FUNCTION_BLOCK Recipe_10058_RedOne
VAR_INPUT
	execute: BOOL;
	Order: DUT_RECIPEORDER;
END_VAR
VAR_OUTPUT
	RecipeInfo: DUT_RECIPEOFFER;
	RecipeDone: BOOL;
	InitDone: BOOL;
	Ready: BOOL;
END_VAR
VAR
	userparametersum: LREAL;
	StepDone: BOOL;
	i: INT;
	Command: ARRAY[1..5] OF DUT_RecipeCommand;
	NextSkill: BOOL;
	SectionReady: BOOL;
END_VAR

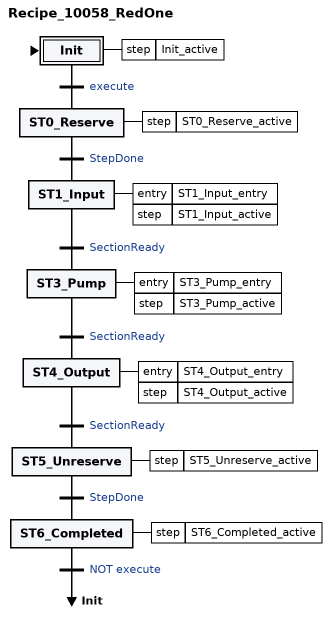
INITIAL_STEP Init:
    Init_active(N);  // step action
END_STEP
TRANSITION FROM Init TO ST0_Reserve
    := execute;
END_TRANSITION
STEP ST0_Reserve:
    ST0_Reserve_active(N);  // step action
END_STEP
TRANSITION FROM ST0_Reserve TO ST1_Input
    := StepDone;
END_TRANSITION
STEP ST1_Input:
    ST1_Input_entry(P1);  // entry action
    ST1_Input_active(N);  // step action
END_STEP
TRANSITION FROM ST1_Input TO ST3_Pump
    := SectionReady;
END_TRANSITION
STEP ST3_Pump:
    ST3_Pump_entry(P1);  // entry action
    ST3_Pump_active(N);  // step action
END_STEP
TRANSITION FROM ST3_Pump TO ST4_Output
    := SectionReady;
END_TRANSITION
STEP ST4_Output:
    ST4_Output_entry(P1);  // entry action
    ST4_Output_active(N);  // step action
END_STEP
TRANSITION FROM ST4_Output TO ST5_Unreserve
    := SectionReady;
END_TRANSITION
STEP ST5_Unreserve:
    ST5_Unreserve_active(N);  // step action
END_STEP
TRANSITION FROM ST5_Unreserve TO ST6_Completed
    := StepDone;
END_TRANSITION
STEP ST6_Completed:
    ST6_Completed_active(N);  // step action
END_STEP
TRANSITION FROM ST6_Completed TO Init
    := NOT execute;
END_TRANSITION

ACTION ST14_Exit_active:
SectionReady := TRUE;
END_ACTION

ACTION ST12_Input_active:
//RT: 2014.11.23: Input Modul auslösen
StepDone := FALSE;

//Skill auswählen
ExecuteSkill.SkillID 		:= 1402;
ExecuteSkill.SkillName	 	:= 'Input';

//Parameter setzen

ExecuteSkill.Parameter[1].ID := 1;
ExecuteSkill.Parameter[1].Name := 'TaskID';
ExecuteSkill.Parameter[1].Value := Order.TaskID;


(*
ExecuteSkill.Parameter[2].ID := ;
ExecuteSkill.Parameter[2].Name := '';
ExecuteSkill.Parameter[2].Value := ;
*)

(*
ExecuteSkill.Parameter[3].ID := ;
ExecuteSkill.Parameter[3].Name := '';
ExecuteSkill.Parameter[3].Value := ;
*)

(*
ExecuteSkill.Parameter[4].ID := ;
ExecuteSkill.Parameter[4].Name := '';
ExecuteSkill.Parameter[4].Value := ;
*)

(*
ExecuteSkill.Parameter[5].ID := ;
ExecuteSkill.Parameter[5].Name := '';
ExecuteSkill.Parameter[5].Value := ;
*)



ExecuteSkill();

StepDone := ExecuteSkill.Done;
END_ACTION

ACTION ST34_Exit_active:
SectionReady := TRUE;
END_ACTION

ACTION ST41_BlockOutput_active:
//RT: 2014.11.23: Blockirt den Mover an Position
StepDone := FALSE;

//Skill auswählen
ExecuteSkill.SkillID 		:= 1315;
ExecuteSkill.SkillName	 	:= 'Block';

//Parameter setzen

ExecuteSkill.Parameter[1].ID := 1;
ExecuteSkill.Parameter[1].Name := 'TaskID';
ExecuteSkill.Parameter[1].Value := Order.TaskID;


(*
ExecuteSkill.Parameter[2].ID := ;
ExecuteSkill.Parameter[2].Name := '';
ExecuteSkill.Parameter[2].Value := ;
*)

(*
ExecuteSkill.Parameter[3].ID := ;
ExecuteSkill.Parameter[3].Name := '';
ExecuteSkill.Parameter[3].Value := ;
*)

(*
ExecuteSkill.Parameter[4].ID := ;
ExecuteSkill.Parameter[4].Name := '';
ExecuteSkill.Parameter[4].Value := ;
*)

(*
ExecuteSkill.Parameter[5].ID := ;
ExecuteSkill.Parameter[5].Name := '';
ExecuteSkill.Parameter[5].Value := ;
*)



ExecuteSkill();

StepDone := ExecuteSkill.Done;
END_ACTION

ACTION ST13_UnblockInput_active:
//RT: 2014.11.23: Gibt Mover Position Frei
StepDone := FALSE;

//Skill auswählen
ExecuteSkill.SkillID 		:= 1316;
ExecuteSkill.SkillName	 	:= 'Unblock';

//Parameter setzen

ExecuteSkill.Parameter[1].ID := 1;
ExecuteSkill.Parameter[1].Name := 'TaskID';
ExecuteSkill.Parameter[1].Value := Order.TaskID;


(*
ExecuteSkill.Parameter[2].ID := ;
ExecuteSkill.Parameter[2].Name := '';
ExecuteSkill.Parameter[2].Value := ;
*)

(*
ExecuteSkill.Parameter[3].ID := ;
ExecuteSkill.Parameter[3].Name := '';
ExecuteSkill.Parameter[3].Value := ;
*)

(*
ExecuteSkill.Parameter[4].ID := ;
ExecuteSkill.Parameter[4].Name := '';
ExecuteSkill.Parameter[4].Value := ;
*)

(*
ExecuteSkill.Parameter[5].ID := ;
ExecuteSkill.Parameter[5].Name := '';
ExecuteSkill.Parameter[5].Value := ;
*)



ExecuteSkill();

StepDone := ExecuteSkill.Done;
END_ACTION

ACTION ST4_Output_active:
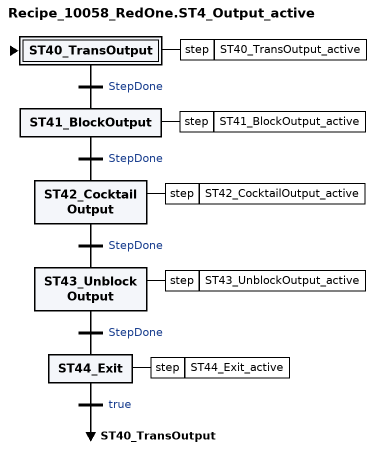
INITIAL_STEP ST40_TransOutput:
    ST40_TransOutput_active(N);  // step action
END_STEP
TRANSITION FROM ST40_TransOutput TO ST41_BlockOutput
    := StepDone;
END_TRANSITION
STEP ST41_BlockOutput:
    ST41_BlockOutput_active(N);  // step action
END_STEP
TRANSITION FROM ST41_BlockOutput TO ST42_CocktailOutput
    := StepDone;
END_TRANSITION
STEP ST42_CocktailOutput:
    ST42_CocktailOutput_active(N);  // step action
END_STEP
TRANSITION FROM ST42_CocktailOutput TO ST43_UnblockOutput
    := StepDone;
END_TRANSITION
STEP ST43_UnblockOutput:
    ST43_UnblockOutput_active(N);  // step action
END_STEP
TRANSITION FROM ST43_UnblockOutput TO ST44_Exit
    := StepDone;
END_TRANSITION
STEP ST44_Exit:
    ST44_Exit_active(N);  // step action
END_STEP
TRANSITION FROM ST44_Exit TO ST40_TransOutput
    := true;
END_TRANSITION
END_ACTION

ACTION ST42_CocktailOutput_active:
//RT: 2014.11.23: Ausgeben des Produktes
StepDone := FALSE;

//Skill auswählen
ExecuteSkill.SkillID 		:= 1403;
ExecuteSkill.SkillName	 	:= 'Output';

//Parameter setzen

ExecuteSkill.Parameter[1].ID := 1;
ExecuteSkill.Parameter[1].Name := 'TaskID';
ExecuteSkill.Parameter[1].Value := Order.TaskID;


(*
ExecuteSkill.Parameter[2].ID := ;
ExecuteSkill.Parameter[2].Name := '';
ExecuteSkill.Parameter[2].Value := ;
*)

(*
ExecuteSkill.Parameter[3].ID := ;
ExecuteSkill.Parameter[3].Name := '';
ExecuteSkill.Parameter[3].Value := ;
*)

(*
ExecuteSkill.Parameter[4].ID := ;
ExecuteSkill.Parameter[4].Name := '';
ExecuteSkill.Parameter[4].Value := ;
*)

(*
ExecuteSkill.Parameter[5].ID := ;
ExecuteSkill.Parameter[5].Name := '';
ExecuteSkill.Parameter[5].Value := ;
*)



ExecuteSkill();

StepDone := ExecuteSkill.Done;
END_ACTION

ACTION ST40_TransOutput_active:
//RT: 2014.11.23: Mover zum Output
StepDone := FALSE;

//Skill auswählen
ExecuteSkill.SkillID 		:= 1320;
ExecuteSkill.SkillName	 	:= 'Transport';

//Parameter setzen

ExecuteSkill.Parameter[3].ID := 3;
ExecuteSkill.Parameter[3].Name := 'Velocity';
ExecuteSkill.Parameter[3].Value := 300;



ExecuteSkill.Parameter[1].ID :=  1;
ExecuteSkill.Parameter[1].Name := 'TargetPosition X';
ExecuteSkill.Parameter[1].Value := 30 ;
ExecuteSkill.Parameter[1].StringValue := '#DP#2#XPosition';



ExecuteSkill.Parameter[2].ID := 2;
ExecuteSkill.Parameter[2].Name := 'TargetPosition Z';
ExecuteSkill.Parameter[2].Value := 100;// ZCookieModule - ZCookieModuleCalibration - 2* Cookiethickness + toppingthickness+ Preasureheight  ;



(* ExecuteSkill.Parameter[4].ID := 4;
ExecuteSkill.Parameter[4].Name := 'Acceleration';
ExecuteSkill.Parameter[4].Value :=0 ;

*)
(*
ExecuteSkill.Parameter[5].ID := ;
ExecuteSkill.Parameter[5].Name := '';
ExecuteSkill.Parameter[5].Value := ;
*)



ExecuteSkill();

StepDone := ExecuteSkill.Done;
END_ACTION

ACTION ST3_Pump_active:
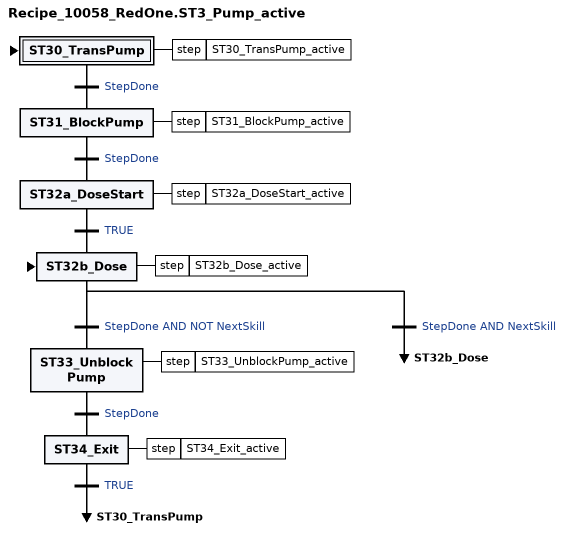
INITIAL_STEP ST30_TransPump:
    ST30_TransPump_active(N);  // step action
END_STEP
TRANSITION FROM ST30_TransPump TO ST31_BlockPump
    := StepDone;
END_TRANSITION
STEP ST31_BlockPump:
    ST31_BlockPump_active(N);  // step action
END_STEP
TRANSITION FROM ST31_BlockPump TO ST32a_DoseStart
    := StepDone;
END_TRANSITION
STEP ST32a_DoseStart:
    ST32a_DoseStart_active(N);  // step action
END_STEP
TRANSITION FROM ST32a_DoseStart TO ST32b_Dose
    := TRUE;
END_TRANSITION
STEP ST32b_Dose:
    ST32b_Dose_active(N);  // step action
END_STEP
TRANSITION FROM ST32b_Dose TO ST33_UnblockPump
    := StepDone AND NOT NextSkill;
END_TRANSITION
STEP ST33_UnblockPump:
    ST33_UnblockPump_active(N);  // step action
END_STEP
TRANSITION FROM ST33_UnblockPump TO ST34_Exit
    := StepDone;
END_TRANSITION
STEP ST34_Exit:
    ST34_Exit_active(N);  // step action
END_STEP
TRANSITION FROM ST34_Exit TO ST30_TransPump
    := TRUE;
END_TRANSITION
TRANSITION FROM ST32b_Dose TO ST32b_Dose
    := StepDone AND NextSkill;
END_TRANSITION
END_ACTION

ACTION ST32a_DoseStart_active:
//RT: 2014.11.23: Summe aller zutaten zum Normiren

userparametersum := 0;
FOR i := 1 TO UserParameterCnt DO
	IF NOT (order.UserParameter[i].Value = 0) THEN
		userparametersum := userparametersum + order.UserParameter[i].Value;
	
	END_IF
END_FOR
IF userparametersum = 0 THEN
userparametersum := -1;
END_IF

//RT: 2014.11.23: Start wert des Arrays setzen
i := 1;
NextSkill := TRUE ;
END_ACTION

ACTION Init_active:
//RT: 2014.11.23: Vorbereiten der daten und der HMI
RecipeDone := FALSE;

// Initialisation of Recipe Parameters an name etc
RecipeInfo.Name := 'Red One';
RecipeInfo.Description := '';
RecipeInfo.Dummy := FALSE;
RecipeInfo.RecipeID := 10058; 	// 
Initdone := TRUE;

//RT: 2014.11.23: wenn weniger als 5 alle lehren skills SkillID := 0
Command[1].SkillID := 1117;
Command[1].SkillName := 'Orange Juice';
Command[1].Quantity := 41;

Command[2].SkillID := 1112;
Command[2].SkillName := 'Lemon Juice';
Command[2].Quantity := 8;

Command[3].SkillID := 1114;
Command[3].SkillName := 'Pineapple Juice';
Command[3].Quantity := 41;

Command[4].SkillID := 1111;
Command[4].SkillName := 'Grenadine Syrup';
Command[4].Quantity := 8;

Command[5].SkillID := 0;
Command[5].SkillName := 'Nothing';
Command[5].Quantity := 0;








//Parameter 0:

	RecipeInfo.UserParameter[0].Dummy 		:= FALSE;
	RecipeInfo.UserParameter[0].Default		:= 200;
	RecipeInfo.UserParameter[0].Description	:= 'Gives the total fluid amount in the glass';
	RecipeInfo.UserParameter[0].MaxValue	:= 200;
	RecipeInfo.UserParameter[0].MinValue	:= 10;
	RecipeInfo.UserParameter[0].Name		:= 'Total Liquid Amount';
	RecipeInfo.UserParameter[0].Unit		:= 'ml';
	
//Parameter 1-5:
FOR i := 1 TO 5 DO
	IF Command[i].SkillID = 0 THEN
		RecipeInfo.UserParameter[i].Dummy 		:= TRUE;
	ELSE
		RecipeInfo.UserParameter[i].Dummy 		:= FALSE;
		RecipeInfo.UserParameter[i].Default		:= Command[i].Quantity;
		RecipeInfo.UserParameter[i].Description	:= Command[i].SkillName;
		RecipeInfo.UserParameter[i].MaxValue	:= 100;
		RecipeInfo.UserParameter[i].MinValue	:= 1;
		RecipeInfo.UserParameter[i].Name		:= Command[i].SkillName;
		RecipeInfo.UserParameter[i].Unit		:= 'ml';	
	END_IF
END_FOR
END_ACTION

ACTION ST30_TransPump_active:
//RT: 2014.11.23: Mover zum Pump
StepDone := FALSE;

//Skill auswählen
ExecuteSkill.SkillID 		:= 1320;
ExecuteSkill.SkillName	 	:= 'Transport';

//Parameter setzen

ExecuteSkill.Parameter[3].ID := 3;
ExecuteSkill.Parameter[3].Name := 'Velocity';
ExecuteSkill.Parameter[3].Value := 1000;



ExecuteSkill.Parameter[1].ID :=  1;
ExecuteSkill.Parameter[1].Name := 'TargetPosition X';
ExecuteSkill.Parameter[1].Value := 30 ;
ExecuteSkill.Parameter[1].StringValue := '#DP#2#XPosition';



ExecuteSkill.Parameter[2].ID := 2;
ExecuteSkill.Parameter[2].Name := 'TargetPosition Z';
ExecuteSkill.Parameter[2].Value := 10;// ZCookieModule - ZCookieModuleCalibration - 2* Cookiethickness + toppingthickness+ Preasureheight  ;



(*
ExecuteSkill.Parameter[4].ID := 4;
ExecuteSkill.Parameter[4].Name := 'Acceleration';
ExecuteSkill.Parameter[4].Value := 0 ;
*)

(*
ExecuteSkill.Parameter[5].ID := ;
ExecuteSkill.Parameter[5].Name := '';
ExecuteSkill.Parameter[5].Value := ;
*)



ExecuteSkill();

StepDone := ExecuteSkill.Done;
END_ACTION

ACTION ST44_Exit_active:
SectionReady := TRUE;
END_ACTION

ACTION ST6_Completed_active:
//RT: 2014.11.23: Warte auf Execute = False
RecipeDone := TRUE;
StepDone := FALSE;
END_ACTION

ACTION ST11_BlockInput_active:
//RT: 2014.11.23: Blockirt den Mover an Position
StepDone := FALSE;

//Skill auswählen
ExecuteSkill.SkillID 		:= 1315;
ExecuteSkill.SkillName	 	:= 'Block';

//Parameter setzen

ExecuteSkill.Parameter[1].ID := 1;
ExecuteSkill.Parameter[1].Name := 'TaskID';
ExecuteSkill.Parameter[1].Value := Order.TaskID;


(*
ExecuteSkill.Parameter[2].ID := ;
ExecuteSkill.Parameter[2].Name := '';
ExecuteSkill.Parameter[2].Value := ;
*)

(*
ExecuteSkill.Parameter[3].ID := ;
ExecuteSkill.Parameter[3].Name := '';
ExecuteSkill.Parameter[3].Value := ;
*)

(*
ExecuteSkill.Parameter[4].ID := ;
ExecuteSkill.Parameter[4].Name := '';
ExecuteSkill.Parameter[4].Value := ;
*)

(*
ExecuteSkill.Parameter[5].ID := ;
ExecuteSkill.Parameter[5].Name := '';
ExecuteSkill.Parameter[5].Value := ;
*)



ExecuteSkill();

StepDone := ExecuteSkill.Done;
END_ACTION

ACTION ST32b_Dose_exit:

END_ACTION

ACTION ST1_Reserve0_active:
//RT: 2014.11.23: Reservire einen Mover

StepDone := FALSE;
RecipeDone := FALSE;
//Skill auswählen
ExecuteSkill.SkillID 		:= 1310;
ExecuteSkill.SkillName	 	:= 'Reserve';

//Parameter setzen

ExecuteSkill.Parameter[1].ID := 1;
ExecuteSkill.Parameter[1].Name := 'TaskID';
ExecuteSkill.Parameter[1].Value := Order.TaskID;

(*
ExecuteSkill.Parameter[2].ID := ;
ExecuteSkill.Parameter[2].Name := '';
ExecuteSkill.Parameter[2].Value := ;
*)

(*
ExecuteSkill.Parameter[3].ID := ;
ExecuteSkill.Parameter[3].Name := '';
ExecuteSkill.Parameter[3].Value := ;
*)

(*
ExecuteSkill.Parameter[4].ID := ;
ExecuteSkill.Parameter[4].Name := '';
ExecuteSkill.Parameter[4].Value := ;
*)

(*
ExecuteSkill.Parameter[5].ID := ;
ExecuteSkill.Parameter[5].Name := '';
ExecuteSkill.Parameter[5].Value := ;
*)

ExecuteSkill();

StepDone := ExecuteSkill.Done;
END_ACTION

ACTION ST33_UnblockPump_active:
//RT: 2014.11.23: Gibt Mover Position Frei
StepDone := FALSE;

//Skill auswählen
ExecuteSkill.SkillID 		:= 1316;
ExecuteSkill.SkillName	 	:= 'Unblock';

//Parameter setzen

ExecuteSkill.Parameter[1].ID := 1;
ExecuteSkill.Parameter[1].Name := 'TaskID';
ExecuteSkill.Parameter[1].Value := Order.TaskID;


(*
ExecuteSkill.Parameter[2].ID := ;
ExecuteSkill.Parameter[2].Name := '';
ExecuteSkill.Parameter[2].Value := ;
*)

(*
ExecuteSkill.Parameter[3].ID := ;
ExecuteSkill.Parameter[3].Name := '';
ExecuteSkill.Parameter[3].Value := ;
*)

(*
ExecuteSkill.Parameter[4].ID := ;
ExecuteSkill.Parameter[4].Name := '';
ExecuteSkill.Parameter[4].Value := ;
*)

(*
ExecuteSkill.Parameter[5].ID := ;
ExecuteSkill.Parameter[5].Name := '';
ExecuteSkill.Parameter[5].Value := ;
*)



ExecuteSkill();

StepDone := ExecuteSkill.Done;
END_ACTION

ACTION ST32b_Dose_active:
//RT: 2014.11.23: Die Dosir Skills anlegen
StepDone := FALSE;

//Skill auswählen
ExecuteSkill.SkillID 		:= Command[i].SkillID;
ExecuteSkill.SkillName	 	:= Command[i].SkillName;
//Parameter setzen

ExecuteSkill.Parameter[0].ID := 1;
ExecuteSkill.Parameter[0].Name := 'Quantity';
//order.userParameter[0] = amount
ExecuteSkill.Parameter[0].Value := order.UserParameter[0].Value * order.UserParameter[i].Value / userparametersum ;//Summe aller Zutatenmengen;

(*
ExecuteSkill.Parameter[2].ID := ;
ExecuteSkill.Parameter[2].Name := '';
ExecuteSkill.Parameter[2].Value := ;
*)

(*
ExecuteSkill.Parameter[3].ID := ;
ExecuteSkill.Parameter[3].Name := '';
ExecuteSkill.Parameter[3].Value := ;
*)

(*
ExecuteSkill.Parameter[4].ID := ;
ExecuteSkill.Parameter[4].Name := '';
ExecuteSkill.Parameter[4].Value := ;
*)

(*
ExecuteSkill.Parameter[5].ID := ;
ExecuteSkill.Parameter[5].Name := '';
ExecuteSkill.Parameter[5].Value := ;
*)


ExecuteSkill();

StepDone := ExecuteSkill.Done;

i := i + 1 ;

IF i = 6 THEN
	NextSkill := FALSE;
ELSIF Command[i].SkillID = 0 THEN
	NextSkill := FALSE;
ELSE
	NextSkill := TRUE;
END_IF
END_ACTION

ACTION ST4_Output_entry:
SectionReady := FALSE;
END_ACTION

ACTION ST3_Pump_entry:
SectionReady := FALSE;
END_ACTION

ACTION ST5_Unreserve_active:
//RT: 2014.11.23: Mover Freigeben
StepDone := FALSE;

//Skill auswählen
ExecuteSkill.SkillID 		:= 1311;
ExecuteSkill.SkillName	 	:= 'Unreserve';

//Parameter setzen

ExecuteSkill.Parameter[1].ID := 1;
ExecuteSkill.Parameter[1].Name := 'TaskID';
ExecuteSkill.Parameter[1].Value := Order.TaskID;


(*
ExecuteSkill.Parameter[2].ID := ;
ExecuteSkill.Parameter[2].Name := '';
ExecuteSkill.Parameter[2].Val ue := ;
*)

(*
ExecuteSkill.Parameter[3].ID := ;
ExecuteSkill.Parameter[3].Name := '';
ExecuteSkill.Parameter[3].Value := ;
*)

(*
ExecuteSkill.Parameter[4].ID := ;
ExecuteSkill.Parameter[4].Name := '';
ExecuteSkill.Parameter[4].Value := ;
*)

(*
ExecuteSkill.Parameter[5].ID := ;
ExecuteSkill.Parameter[5].Name := '';
ExecuteSkill.Parameter[5].Value := ;
*)



ExecuteSkill();

StepDone := ExecuteSkill.Done;
END_ACTION

ACTION ST1_Input_active:
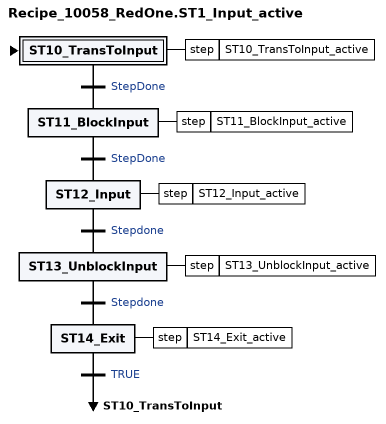
INITIAL_STEP ST10_TransToInput:
    ST10_TransToInput_active(N);  // step action
END_STEP
TRANSITION FROM ST10_TransToInput TO ST11_BlockInput
    := StepDone;
END_TRANSITION
STEP ST11_BlockInput:
    ST11_BlockInput_active(N);  // step action
END_STEP
TRANSITION FROM ST11_BlockInput TO ST12_Input
    := StepDone;
END_TRANSITION
STEP ST12_Input:
    ST12_Input_active(N);  // step action
END_STEP
TRANSITION FROM ST12_Input TO ST13_UnblockInput
    := Stepdone;
END_TRANSITION
STEP ST13_UnblockInput:
    ST13_UnblockInput_active(N);  // step action
END_STEP
TRANSITION FROM ST13_UnblockInput TO ST14_Exit
    := Stepdone;
END_TRANSITION
STEP ST14_Exit:
    ST14_Exit_active(N);  // step action
END_STEP
TRANSITION FROM ST14_Exit TO ST10_TransToInput
    := TRUE;
END_TRANSITION
END_ACTION

ACTION ST43_UnblockOutput_active:
//RT: 2014.11.23: Gibt Mover Position Frei
StepDone := FALSE;

//Skill auswählen
ExecuteSkill.SkillID 		:= 1316;
ExecuteSkill.SkillName	 	:= 'Unblock';

//Parameter setzen

ExecuteSkill.Parameter[1].ID := 1;
ExecuteSkill.Parameter[1].Name := 'TaskID';
ExecuteSkill.Parameter[1].Value := Order.TaskID;


(*
ExecuteSkill.Parameter[2].ID := ;
ExecuteSkill.Parameter[2].Name := '';
ExecuteSkill.Parameter[2].Value := ;
*)

(*
ExecuteSkill.Parameter[3].ID := ;
ExecuteSkill.Parameter[3].Name := '';
ExecuteSkill.Parameter[3].Value := ;
*)

(*
ExecuteSkill.Parameter[4].ID := ;
ExecuteSkill.Parameter[4].Name := '';
ExecuteSkill.Parameter[4].Value := ;
*)

(*
ExecuteSkill.Parameter[5].ID := ;
ExecuteSkill.Parameter[5].Name := '';
ExecuteSkill.Parameter[5].Value := ;
*)



ExecuteSkill();

StepDone := ExecuteSkill.Done;
END_ACTION

ACTION ST0_Reserve_active:
//RT: 2014.11.23: Reservire einen Mover

StepDone := FALSE;
RecipeDone := FALSE;
//Skill auswählen
ExecuteSkill.SkillID 		:= 1310;
ExecuteSkill.SkillName	 	:= 'Reserve';

//Parameter setzen

ExecuteSkill.Parameter[1].ID := 1;
ExecuteSkill.Parameter[1].Name := 'TaskID';
ExecuteSkill.Parameter[1].Value := Order.TaskID;

(*
ExecuteSkill.Parameter[2].ID := ;
ExecuteSkill.Parameter[2].Name := '';
ExecuteSkill.Parameter[2].Value := ;
*)

(*
ExecuteSkill.Parameter[3].ID := ;
ExecuteSkill.Parameter[3].Name := '';
ExecuteSkill.Parameter[3].Value := ;
*)

(*
ExecuteSkill.Parameter[4].ID := ;
ExecuteSkill.Parameter[4].Name := '';
ExecuteSkill.Parameter[4].Value := ;
*)

(*
ExecuteSkill.Parameter[5].ID := ;
ExecuteSkill.Parameter[5].Name := '';
ExecuteSkill.Parameter[5].Value := ;
*)

ExecuteSkill();

StepDone := ExecuteSkill.Done;
END_ACTION

ACTION ST1_Input_entry:
SectionReady := FALSE;
END_ACTION

ACTION ST10_TransToInput_active:
//RT: 2014.11.23: Mover zum Input

StepDone := FALSE;

//Skill auswählen
ExecuteSkill.SkillID 		:= 1320;
ExecuteSkill.SkillName	 	:= 'Transport';

//Parameter setzen

ExecuteSkill.Parameter[3].ID := 3;
ExecuteSkill.Parameter[3].Name := 'Velocity';
ExecuteSkill.Parameter[3].Value := 1000;



ExecuteSkill.Parameter[1].ID :=  1;
ExecuteSkill.Parameter[1].Name := 'TargetPosition X';
ExecuteSkill.Parameter[1].Value := 30 ;
ExecuteSkill.Parameter[1].StringValue := '#DP#2#XPosition';



ExecuteSkill.Parameter[2].ID := 2;
ExecuteSkill.Parameter[2].Name := 'TargetPosition Z';
ExecuteSkill.Parameter[2].Value := 100;// ZCookieModule - ZCookieModuleCalibration - 2* Cookiethickness + toppingthickness+ Preasureheight  ;



(*
ExecuteSkill.Parameter[4].ID := 4;
ExecuteSkill.Parameter[4].Name := 'Acceleration';
ExecuteSkill.Parameter[4].Value := 0 ;
*)

(*
ExecuteSkill.Parameter[5].ID := ;
ExecuteSkill.Parameter[5].Name := '';
ExecuteSkill.Parameter[5].Value := ;
*)



ExecuteSkill();

StepDone := ExecuteSkill.Done;
END_ACTION

ACTION ST31_BlockPump_active:
//RT: 2014.11.23: Blockirt den Mover an Position
StepDone := FALSE;

//Skill auswählen
ExecuteSkill.SkillID 		:= 1315;
ExecuteSkill.SkillName	 	:= 'Block';

//Parameter setzen

ExecuteSkill.Parameter[1].ID := 1;
ExecuteSkill.Parameter[1].Name := 'TaskID';
ExecuteSkill.Parameter[1].Value := Order.TaskID;


(*
ExecuteSkill.Parameter[2].ID := ;
ExecuteSkill.Parameter[2].Name := '';
ExecuteSkill.Parameter[2].Value := ;
*)

(*
ExecuteSkill.Parameter[3].ID := ;
ExecuteSkill.Parameter[3].Name := '';
ExecuteSkill.Parameter[3].Value := ;
*)

(*
ExecuteSkill.Parameter[4].ID := ;
ExecuteSkill.Parameter[4].Name := '';
ExecuteSkill.Parameter[4].Value := ;
*)

(*
ExecuteSkill.Parameter[5].ID := ;
ExecuteSkill.Parameter[5].Name := '';
ExecuteSkill.Parameter[5].Value := ;
*)



ExecuteSkill();

StepDone := ExecuteSkill.Done;
END_ACTION

END_FUNCTION_BLOCK

(* stored: Version 1.1.0.1, ProductVersion 3.1.0.25
   POU Recipe_10058_RedOne: Id {2c064201-8a5c-49ce-acee-d6ca01fb923b}
   Action ST14_Exit_active: Id {0863dcc2-0557-4861-aff6-37a039ca2718}
   Action ST12_Input_active: Id {0aceb5f3-5424-4081-a964-818bfb68fd9e}
   Action ST34_Exit_active: Id {120a63a5-93a7-4747-be88-b9ef95a29875}
   Action ST41_BlockOutput_active: Id {2b83f0b1-64d7-409f-92ad-db318c19800c}
   Action ST13_UnblockInput_active: Id {3030d505-a4de-4564-9cc2-8e514e1f7168}
   Action ST4_Output_active: Id {3039ca4c-6c9c-40bf-8a4a-c39c8ceecadd}
   Action ST42_CocktailOutput_active: Id {333be4fb-404f-44ee-a665-d18fab24d6f8}
   Action ST40_TransOutput_active: Id {3d1605fe-45d7-4ec9-b353-02f5d0f23f50}
   Action ST3_Pump_active: Id {432db1c3-1b03-4a69-96f4-85c4ab6e015e}
   Action ST32a_DoseStart_active: Id {43a53962-0cbb-46ea-9619-f254bfafdab3}
   Action Init_active: Id {58d24451-d898-49da-9f60-92a61089dd3d}
   Action ST30_TransPump_active: Id {6b3ddfc8-5e7f-4bee-99dd-9ff529cd0b35}
   Action ST44_Exit_active: Id {75b2e525-d0fb-4194-94bd-da9867c9bfa2}
   Action ST6_Completed_active: Id {770f06a8-5511-40d4-afb7-669f6bfc3adc}
   Action ST11_BlockInput_active: Id {793e1878-45e6-4c88-93fc-0c627b689fc3}
   Action ST32b_Dose_exit: Id {7afa16e5-7cb7-4984-8cb5-c5dfb3bbe696}
   Action ST1_Reserve0_active: Id {8fb7f144-4cd9-47ff-86bf-e3230bf1fcdc}
   Action ST33_UnblockPump_active: Id {9eae5324-f584-413a-bf24-b63799973d1a}
   Action ST32b_Dose_active: Id {a772fc72-31b7-46b9-afc1-c88680cb74ba}
   Action ST4_Output_entry: Id {ae36edda-9a7d-479f-8d25-b95d8d500c1f}
   Action ST3_Pump_entry: Id {ba13b6bd-f1b2-4239-8778-8fc97c526a50}
   Action ST5_Unreserve_active: Id {c025a216-28a5-472e-b4db-348f54441dd8}
   Action ST1_Input_active: Id {c6c9751d-43e6-469f-80d5-7fb53724dde9}
   Action ST43_UnblockOutput_active: Id {ca0ff69a-3a25-4be0-9a92-a345d8c46191}
   Action ST0_Reserve_active: Id {cdf4ed95-f14a-4bb7-b36e-40adf736b70b}
   Action ST1_Input_entry: Id {d746b80e-85d0-416b-92be-47c6cc9f6bfa}
   Action ST10_TransToInput_active: Id {f1d4295e-b444-4490-a5e0-00fca66b335e}
   Action ST31_BlockPump_active: Id {fd7fba64-0a6c-4280-9351-32bd30318fc4} *)
